TYPE MotorInputVariables :
STRUCT
	Start : BOOL;
	Stop : BOOL;
	Oveload : BOOL;
	
END_STRUCT
END_TYPE

(* stored: Version 1.1.0.1, ProductVersion 3.1.4024.9
   DUT MotorInputVariables: Id {ee07eff9-7f78-46df-926f-fcfdb75fea8a} *)
